Staubli VAL3: main.pgx

public program main()
  local num lKey
begin
end
